{attribute 'call_after_init'}
FUNCTION_BLOCK FB_SafeBPCompare_Test EXTENDS TcUnit.FB_TestSuite
VAR_INPUT
END_VAR
VAR_OUTPUT
END_VAR
VAR

END_VAR

BeamOffIsSafe();
BPComparisonCheck();

//Verify beam off is considered safe.
METHOD BeamOffIsSafe
VAR_INPUT
END_VAR
VAR
	stBeamOn	:	ST_BeamParams;
	stBeamOff	:	ST_BeamParams;
	
END_VAR
stBeamOn := F_SetBeamParams(
	50, //50% attenuation is more conservative than 0
	10,
	16#FFFF,
	120);

stBeamOff := F_SetBeamParams(
	0, //0% attenuation
	10,
	16#FFFF,
	0); //0 beam rate means this bps is actually safer than BeamOn

TEST('BeamOffIsSafe');
	
AssertTrue(
	F_SafeBPCompare(stBeamOff, stBeamOn),
	'SafeBPCompare does not think beam rate = 0 is safer than anything else.'); 
TEST_FINISHED();
END_METHOD

//Verify BP comparison remains logical.
METHOD BPComparisonCheck
VAR_INPUT
END_VAR
VAR
	stSafer	:	ST_BeamParams;
	stNotSoSafe	:	ST_BeamParams;
END_VAR
TEST('BPComparisonCheck');


//Attenuation
stSafer := F_SetBeamParams(
	1, //
	10,
	16#FFFF,
	1);

stNotSoSafe := F_SetBeamParams(
	0, //
	10,
	16#FFFF,
	1); 
	
AssertTrue(
	F_SafeBPCompare(stSafer, stNotSoSafe),
	'Attenuation eval is broken (True)'); 

AssertFalse(
	F_SafeBPCompare(stNotSoSafe, stSafer),
	'Attenuation eval is broken (False)');
	
	
//Rate
stSafer := F_SetBeamParams(
	0,
	10,
	16#FFFF,
	1); //

stNotSoSafe := F_SetBeamParams(
	0,
	10,
	16#FFFF,
	10); //
	
AssertTrue(
	F_SafeBPCompare(stSafer, stNotSoSafe),
	'Rate eval is broken (True)'); 

AssertFalse(
	F_SafeBPCompare(stNotSoSafe, stSafer),
	'Rate eval is broken (False)');
	
//Pulse energy
stSafer := F_SetBeamParams(
	0, 
	1, //
	16#FFFF,
	1);

stNotSoSafe := F_SetBeamParams(
	0, 
	10, //
	16#FFFF,
	1); 
	
AssertTrue(
	F_SafeBPCompare(stSafer, stNotSoSafe),
	'Pulse energy eval is broken (True)'); 

AssertFalse(
	F_SafeBPCompare(stNotSoSafe, stSafer),
	'Pulse energy eval is broken (False)');	
	
//Photon energy
//More extensive tests elsewhere
stSafer := F_SetBeamParams(
	0, 
	1, 
	2#0000_0000_0000_0110, //200-400eV
	1);
	
stSafer.reV := 300; //

stNotSoSafe := F_SetBeamParams(
	0, 
	1, 
	2#0000_0000_0000_0110, //200-400ev
	1);
	
stNotSoSafe.reV := 401;
	
AssertTrue(
	F_SafeBPCompare(stSafer, stNotSoSafe),
	'Photon energy eval is broken (True)'); 

AssertFalse(
	F_SafeBPCompare(stNotSoSafe, stSafer),
	'Photon energy eval is broken (False)');	
TEST_FINISHED();
END_METHOD

END_FUNCTION_BLOCK

(* stored: Version 1.1.0.1, ProductVersion 3.1.4024.0
   POU FB_SafeBPCompare_Test: Id {8a1c9dec-d419-4671-8e9f-3bf503fe2c8f}, SpecialFunc None
   Method BeamOffIsSafe: Id {baafb4a0-1daf-4334-8116-72ea06a2d1cd}
   Method BPComparisonCheck: Id {204e7277-8e23-4c94-9e2b-614a24b72a02} *)
